# EPICS IOC start-up script: examples/test/PSI/EP7211-0034_AM8111/EP7211-0034_AM8111_CSV.iocsh
require ecmccfg

${SCRIPTEXEC} ${ecmccfg_DIR}configureSlave.cmd, "SLAVE_ID=3, HW_DESC=EP7211-0034, CONFIG=-Motor-Beckhoff-AM8111-0F20-0000"

# Apply hardware configuration
${SCRIPTEXEC} ${ecmccfg_DIR}applyConfig.cmd

epicsEnvSet("DEV",      "STEST-MYDEVICE")
${SCRIPTEXEC} ${ecmccfg_DIR}configureAxis.cmd,            "CONFIG=./cfg/AM8111_CSV.pax"
